// TIA Portal V16 export
// export: Created 2024-12-03T15:41:44.9432173Z, ExportSetting WithReadOnly, DisplayName Totally Integrated Automation Portal, DisplayVersion V16 Update 6, DisplayName TIA Portal Version Control Interface, DisplayVersion V16 Update 2, DisplayName TIA Portal Openness, DisplayVersion V16 Update 6, DisplayName TIA Portal Teamcenter Gateway, DisplayVersion V16, DisplayName SINAMICS Startdrive Advanced, DisplayVersion V16 Update 5, DisplayName SINAMICS Startdrive G130, G150, S120, S150, SINAMICS MV, S210, DisplayVersion V16 Update 5, DisplayName SINAMICS Startdrive G110M, G120, G120C, G120D, G120P, G115D, DisplayVersion V16 Update 5, DisplayName STEP 7 Professional, DisplayVersion V16 Update 6, DisplayName STEP 7 Safety, DisplayVersion V16, DisplayName WinCC Advanced / Unified PC, DisplayVersion V16 Update 6
TYPE "CLXAiPLCmini_IN_UDT"
// stored: CreationDate 2021-07-13T07:41:36.2278727Z, InterfaceModifiedDate 2020-05-02T16:54:33.6185899Z, IsConsistent true, LibraryConformanceStatus The object is library-conformant., ModifiedDate 2021-03-27T07:36:57.0070798Z
   STRUCT
      AllSensors { ExternalVisible := 'False'} : Struct   // All sensor inputs
         "Reserved[0]" : Bool;
         "Reserved[1]" : Bool;
         "Reserved[2]" : Bool;
         "Reserved[3]" : Bool;
         "Reserved[4]" : Bool;
         "Reserved[5]" : Bool;
         "Reserved[6]" : Bool;
         Heartbeat : Bool;   // This bit toggles every 2 seconds .
         LeftPin2 : Bool;   // Left sensor port state (Pin2)
         "Reserved[9]" : Bool;
         RightPin2 : Bool;   // Right sensor port state (Pin2)
         "Reserved[11]" : Bool;
         LeftPin4 : Bool;   // Left sensor port state (Pin4)
         "Reserved[13]" : Bool;
         RightPin4 : Bool;   // Right sensor port state (Pin4)
         "Reserved[15]" : Bool;
      END_STRUCT;
      SensorDetect { ExternalVisible := 'False'} : Struct   // Sensor detection
         Reserved : Byte;
         RightSensorDetect : Bool;   // If this bit is TRUE a sensor has been detected on the Right sensor port
         LeftSensorDetect : Bool;   // If this bit is TRUE a sensor has been detected on the Left sensor port
         "Reserved[10]" : Bool;
         "Reserved[11]" : Bool;
         "Reserved[12]" : Bool;
         "Reserved[13]" : Bool;
         "Reserved[14]" : Bool;
         "Reserved[15]" : Bool;
      END_STRUCT;
      LeftCalcTemp { ExternalVisible := 'False'} : Byte;   // The temperature of the Left MDR in degrees Celsius
      ModuleTemp { ExternalVisible := 'False'} : Byte;   // The temperature of the module in degrees Celsius
      LeftMDRDiagnostic { ExternalVisible := 'False'} : Struct   // Left MDR diagnostics .
         Overheat : Bool;   // The MDR 's temperature has exceeded 105 degrees Celsius
         MaxTorque : Bool;   // The MDR is running with maximum torque output
         ShortCircuit : Bool;   // There is a short circuit on the MDR
         MDRNotConnected : Bool;   // The MDR is not connected
         Overload : Bool;   // The MDR has been overloaded - this means its speed is less than 10% of the selected speed
         Stalled : Bool;   // The MDR has stalled
         MDRBadHall : Bool;   // The MDR has a Hall Efect Sensor error
         MDRNotUsed : Bool;   // The MDR is not used
         MDRStatus1 : Bool;   // This field and the next are used together by the module to indicate the status of the MDR. Please refer to documentation
         MDRStatus2 : Bool;
         MDRinDOmode : Bool;   // The MDR is in digital Output mode .
         Reserved1 : Bool;
         Reserved2 : Bool;
         Reserved3 : Bool;
         OverVoltage : Bool;   // The sum of the module power supply voltage + the MDR-generated voltage has exceeded 30 volts
         LowVoltage : Bool;   // Module power supply is less than 18 Volts
      END_STRUCT;
      RightCalcTemp { ExternalVisible := 'False'} : Byte;   // The temperature of the Right MDR in degrees Celsius
      ModuleTemp_1 { ExternalVisible := 'False'} : Byte;   // The temperature of the module in degrees Celsius
      RightMDRDiagnostic { ExternalVisible := 'False'} : Struct   // Right MDR diagnostics .
         Overheat : Bool;   // The MDR 's temperature has exceeded 105 degrees Celsius
         MaxTorque : Bool;   // The MDR is running with maximum torque output
         ShortCircuit : Bool;   // There is a short circuit on the MDR
         MDRNotConnected : Bool;   // The MDR is not connected
         Overload : Bool;   // The MDR has been overloaded - this means its speed is less than 10% of the selected speed
         Stalled : Bool;   // The MDR has stalled
         MDRBadHall : Bool;   // The MDR has a Hall Efect Sensor error
         MDRNotUsed : Bool;   // The MDR is not used
         MDRStatus1 : Bool;   // This field and the next are used together by the module to indicate the status of the MDR. Please refer to documentation
         MDRStatus2 : Bool;
         MDRinDOmode : Bool;   // The MDR is in digital Output mode .
         Reserved1 : Bool;
         Reserved2 : Bool;
         Reserved3 : Bool;
         OverVoltage : Bool;   // The sum of the module power supply voltage + the MDR-generated voltage has exceeded 30 volts
         LowVoltage : Bool;   // Module power supply is less than 18 Volts
      END_STRUCT;
      LeftMDR_DIOstatus : Struct   // This is the status when the MDR is used as a digital IO
         Reserved0 : Bool;
         Reserved1 : Bool;
         Reserved2 : Bool;
         Reserved3 : Bool;
         ShortCircuit : Bool;   // When this bit is '1' , there is a short circuit between +24V and Pin2/3/4
         Reserved5 : Bool;
         Reserved6 : Bool;
         Reserved7 : Bool;
         Reserved : Byte;
      END_STRUCT;
      RightMDR_DIOstatus : Struct   // This is the status when the MDR is used as a digital IO
         Reserved0 : Bool;
         Reserved1 : Bool;
         Reserved2 : Bool;
         Reserved3 : Bool;
         ShortCircuit : Bool;   // When this bit is '1' , there is a short circuit between +24V and Pin2/3/4
         Reserved5 : Bool;
         Reserved6 : Bool;
         Reserved7 : Bool;
         Reserved : Byte;
      END_STRUCT;
   END_STRUCT;
END_TYPE
